TYPE ST_Alarm :
STRUCT
	sCode							: STRING;
	bIsActive						: BOOL;
	bWrittenOnGeneralAlarm			: BOOL;
END_STRUCT
END_TYPE

(* stored: Version 1.1.0.1
   DUT ST_Alarm: Id {8a549dec-c515-4e84-925c-cf6c515154e4} *)
